(*
SPDX-FileCopyrightText: © 2026 Oleksandr Tiutyk <trofimich@gmail.com>
SPDX-License-Identifier: MIT
License: https://opensource.org/license/mit
*)

(*!
<summary>
Beckhoff EL6022: Serial communication channel process image.
</summary>
<description>
Encapsulates 22-byte input (InData) and output (OutData) process data for one RS422/RS485 communication
channel.
When used for I/O, link located fields or their containing buffers to the matching selected PDOs.
The record is not a packed wire buffer; compiler padding is not part of the device specification.
Unlinked/default values do not prove valid I/O. The caller evaluates bus/channel validity before use.
Use one owner task per instance and externally synchronize other access; multi-field snapshots are not atomic.
Copies store data without creating hardware links. Keep borrowed field references valid while consumers are bound.
This passive record performs no validation, synchronization, configuration or protocol advancement.
Select the 22-byte serial payload with 16-bit status/control words; larger buffers and 9-bit modes
are outside this model. The owning service implements the transmit/receive toggle handshake.
</description>
*)
TYPE EL6022_CHANNEL :
STRUCT
	InData AT %I* : EL6xxx22ByteInData;
	OutData AT %Q* : EL6xxx22ByteOutData;
END_STRUCT
END_TYPE

(* stored: Version 1.1.0.1, ProductVersion 3.1.4026.18
   DUT EL6022_CHANNEL: Id {36e66333-6d37-4900-88c9-78bd5358e8ea} *)
